FUNCTION_BLOCK FB_AllInOne
VAR_INPUT
	ParamNameAllInOne		: STRING 	:= 'Wind spd + dir + hygro + temp';				// (NA) Name of the pyranometer : to easily identify it
	ParamTempoComAlarm		: TIME 		:= T#10S ; 										// (s) Config : Tempo to detect LOC Alarm
	{attribute 'OPC.UA.DA' := '1'} 
	ParamClockReadTime 		: TIME 		:= T#2S;	  									// (Time) Read Modbus Frequency . 
 	ParamTimeout			: TIME  	:= T#5S ;		  								// (Time) Timeout for modbus reading
	{attribute 'OPC.UA.DA' := '1'} 
	ParamUnitID				: BYTE		:= 1;											// (NA) Unit ID for modbus reading
	{attribute 'OPC.UA.DA' := '1'} 
	ParamTCPPort			: UINT		:= 502;											// (NA) TCP port for modbus
	{attribute 'OPC.UA.DA' := '1'} 
	ParamIpAddress			: STRING	:= '127.0.0.1';									// (NA) IP address for modbus
END_VAR

VAR
	//M_AlarmManagement
	TON_ComAlarm				: TON ; 								// Tempo before deteting loss of communication. 

	
	IN_CmdReset_L					: BOOL;                                                        	
		
	// M_READ VARIABLES//
MesData		AT %Q*  : AllInOne ; 							// (NA) [P,H,B] INV  Data Structure 
	FB_ModbusReadInputRegs		: ARRAY[1..2] OF FB_MBReadInputRegs;	// FB for Modbus Read
	MesBlock1_Temp 				: ARRAY[1..96]  OF WORD; 				// (NA) Temporary Block with multiple modbus reading (Caution : Double Word variables)
	MesBlock2_Temp 				: ARRAY[1..3]  OF WORD; 				// (NA) Temporary Block with multiple modbus reading (Caution : Double Word variables)
	MesModbusReadAlarm1 		: BOOL ; 								// (NA) Modbus Read Alarm for all modbus frames		
	MesModbusReadAlarm2 		: BOOL ; 								// (NA) Modbus Read Alarm for all modbus frames		
	MesAlarmCom					: BOOL;                         		
	MesModbusAlarmCode			: UDINT;								// (NA) Modbus Read Alarm Code	
	                                                            		
	// M_STATEMANAGER//                                         		
	FB_OperationIndex			: FB_OperationIndex ;           		
	MesLastStart				: STRING ;			 					// Datetime of the last Start
	MesState					: BYTE ; 								// (NA) Cal                                                                                                            	
	MesRunningTime				: INT ; 								// Total Running Time
	                                                        			
	//M_EXECUTE VARIABLES //                                		
	TP1							: TP ; 									// (NA) Tempo to define Modbus Reading Frequency 
	                                                        	
	ClockRead				AT %Q*	: BOOL;								// (NA) Modbus reading Clock
	
	
	//M_INIT //
	bInit 						: BOOL;							 
END_VAR

VAR_OUTPUT
END_VAR
VAR
END_VAR

METHOD M_AlarmManagement
//////////////////
// Manages IntelliGen Alarms
/////////////////

VAR 
	// Method local variables (reinitialized at each cycle) 
	FB_AlarmCodeManager : FB_AlarmCodeManager ; 
END_VAR

TON_ComAlarm(IN:= (MesModbusReadAlarm1) AND (MesModbusReadAlarm2) , PT:= ParamTempoComAlarm, Q=>MesAlarmCom) ;	

FB_AlarmCodeManager(
		bAlarm1			:= MesAlarmCom,  					// No connexion to inverter 
		bAlarm2			:= FALSE,//
		bAlarm3			:= False,//
		bAlarm4			:= False,//
		bAlarm5			:= False,//
		bAlarm6			:= FALSE, 							//
		bAlarm7			:= False, 							//
		bAlarm8			:= False, 							//
		bAlarm9			:= False, 							//
		bAlarm10		:= False, 							//
		bAlarm11		:= FALSE,                         //
		bAlarm12		:= FALSE,                         //
		bAlarm13		:= FALSE,                         //
		bAlarm14		:= FALSE, 							// 
		bAlarm15		:= FALSE , 			// 
		wAlarmCode		=>MesData.MesAlarmCode);
END_METHOD

METHOD M_Execute
//////////////////
//  Method Calls 
/////////////////

VAR 
	// Method local variables (reinitialized at each cycle) 

END_VAR
IF NOT bInit THEN
	M_Init();
END_IF

// READING AND WRITING CLOCK //
	TP1(IN:=NOT TP1.Q , PT:= ParamClockReadTime);
	ClockRead 				:= TP1.Q;
	
	

// METHODS CALLS//
	M_Read();



	/////////
	M_StateManager() ; 
	

	M_AlarmManagement();
END_METHOD

METHOD M_Init : BOOL
VAR_INPUT
END_VAR


bInit := FALSE;
END_METHOD

{attribute 'object_name' := 'M_Read'}
METHOD M_Read
//////////
// Read Method for SMA : Modbus reading
//////////
VAR
	// Method local variables (reinitialized at each cycle) 
	MW 					: FB_MergeWordsToDint; 
	tets : uint;
END_VAR

FB_ModbusReadInputRegs[1]
(	
	pDestAddr := ADR(MesBlock1_Temp),
	sIPAddr := ParamIpAddress,
	tTimeout := T#1S,
	nQuantity := 96,
	ntcpport := ParamTCPPort,
	nMBAddr := 0,
	cbLength := 96*2,
	nUnitID := 1,
	bExecute := ClockRead,
	nErrId => MesModbusAlarmCode,
	bError => MesModbusReadAlarm1
);
FB_ModbusReadInputRegs[2]
(	
	pDestAddr := ADR(MesBlock2_Temp),
	sIPAddr := ParamIpAddress,
	tTimeout := T#1S,
	nQuantity := 3,
	ntcpport := ParamTCPPort,
	nMBAddr := 4128,
	cbLength := 3*2,
	nUnitID := 1,
	bExecute := ClockRead,
	nErrId => MesModbusAlarmCode,
	bError => MesModbusReadAlarm2
);
	


	
MW(WORD_STRONG := MesBlock1_Temp[65], size := 1, fix := 1,SIGNED := TRUE, VAR_OUT := MesData.MesTemp_Amb);
MW(WORD_STRONG := MesBlock1_Temp[66], size := 1, fix := 0,SIGNED := FALSE, VAR_OUT := MesData.MesAlarmTemp);
MW(WORD_STRONG := MesBlock1_Temp[3], size := 1, fix := 1,SIGNED := TRUE, VAR_OUT := MesData.MesHygro);
MW(WORD_STRONG := MesBlock1_Temp[4], size := 1, fix := 0,SIGNED := FALSE, VAR_OUT := MesData.MesAlarmHygro);
MW(WORD_STRONG := MesBlock1_Temp[5], size := 1, fix := 1,SIGNED := TRUE, VAR_OUT := MesData.MesDewPoint);
MW(WORD_STRONG := MesBlock1_Temp[6], size := 1, fix := 0,SIGNED := FALSE, VAR_OUT := MesData.MesAlarmDewPt);
MW(WORD_STRONG := MesBlock1_Temp[93], size := 1, fix := 2,SIGNED := TRUE, VAR_OUT := MesData.MesWindSp);
MW(WORD_STRONG := MesBlock1_Temp[94], size := 1, fix := 0,SIGNED := FALSE, VAR_OUT := MesData.MesAlarmWindSp);
MW(WORD_STRONG := MesBlock1_Temp[95], size := 1, fix := 1,SIGNED := TRUE, VAR_OUT := MesData.MesWindDir);
MW(WORD_STRONG := MesBlock1_Temp[96], size := 1, fix := 0,SIGNED := FALSE, VAR_OUT := MesData.MesAlarmWindDir);

	
MW(WORD_STRONG := MesBlock2_Temp[1], size := 1, fix := 0,SIGNED := TRUE, VAR_OUT := MesData.MesRain1);
MW(WORD_STRONG := MesBlock2_Temp[2], size := 1, fix := 0,SIGNED := TRUE, VAR_OUT := MesData.MesRain2);
MW(WORD_STRONG := MesBlock2_Temp[3], size := 1, fix := 0,SIGNED := TRUE, VAR_OUT := MesData.MesRain3);
END_METHOD

METHOD M_StateManager
//////////////////
// Detect which is the state of the inverter. IF loss of communication MesState =0 , the last inverter state is kept .  
/////////////////

VAR 
	// Method local variables (reinitialized at each cycle) 

	
END_VAR
// OPERATIONNAL INDEX //
//	FB_OperationIndex(
//		MesON 				:= MesState>1, 
//		CmdReset 			:= CmdReInitMaintenanceIndicator_G,
//		CalRunningTimeHr 	=> CalRunningTime , 
//		CalNbMove 			=> CalNbMove,
//		CalTimeStart 		=> CalLastStart) ;
END_METHOD

END_FUNCTION_BLOCK

(* stored: Version 1.1.0.1, ProductVersion 3.1.4024.6
   POU FB_AllInOne: Id {a3b88c7a-e1b9-48ec-bd33-0f503332ce50}, SpecialFunc None
   Method M_AlarmManagement: Id {47a45b6f-0724-49ec-8e2e-95599688b294}
   Method M_Execute: Id {b3f87000-892a-4895-bf0d-5f4baa7d1be1}
   Method M_Init: Id {138b198f-455f-4b0b-9f08-49c7d41a30cc}
   Method M_Read: Id {cadf178c-5bd0-4980-81dd-a5eacf4f4ecb}
   Method M_StateManager: Id {c35091d4-452e-4f8f-9dea-9c7c034a7192} *)
